{attribute 'OPC.UA.DA.StructuredType' := '1'}
FUNCTION_BLOCK FB_Unit_RO_RND EXTENDS FB_BaseDevice IMPLEMENTS I_Device

VAR
	bFirstRun: BOOL := TRUE;
	{attribute 'OPC.UA.DA' := '1'} 
	bOutContactor AT %Q*: BOOL := FALSE;
	
	
	{attribute 'OPC.UA.DA' := '0'} 
	eSMState: (WAIT, TURNING_ON, ON, TURNING_OFF, OFF);
	
	tDebounce: TIME := T#5S;
	fbTON_Debounce: TON := (PT := tDebounce, IN := FALSE);
	
END_VAR

fbTON_Debounce();

IF bFirstRun THEN
	fbTON_Debounce.IN := TRUE;
	bFirstRun := FALSE;
END_IF


IF GVL.bAutoUpdateDeviceState THEN
	eState := eStateTarget;	
END_IF


IF eMode = E_DeviceMode.MANUAL THEN
	bEnable := TRUE;
END_IF

IF bEnable AND eStateTarget = E_DeviceState.ON AND eState <> E_DeviceState.ON THEN
		eSMState := TURNING_ON;
END_IF

IF (bEnable = FALSE OR eStateTarget = E_DeviceState.OFF) AND eState <> E_DeviceState.OFF THEN
		eSMState := TURNING_OFF;
END_IF


CASE eSMState OF
	
	WAIT:
		//Wait for method call to change ESMState
		
	TURNING_ON: 
		IF fbTON_Debounce.Q THEN
			eState := E_DeviceState.TURNING_ON;
			bOutContactor := TRUE;
			fbTON_Debounce.IN := FALSE;
			eSMState := ON;
		END_IF

		
	ON:
		IF bOutContactor <> TRUE THEN
			raiseAlarm(Priority := E_AlarmPriority.High, Label := 'Power Lost', Enabled := TRUE, DeviceAlarmID := 1);
			eState := E_DeviceState.OFF;
			eSMState := TURNING_OFF;
		END_IF
			
	TURNING_OFF:
		fbTON_Debounce.IN := TRUE;
		bOutContactor := TRUE;
		eState := E_DeviceState.TURNING_OFF;
		bOutContactor := FALSE;
		eSMState := OFF;

	OFF:
		eState := E_DeviceState.OFF;
		eSMState := WAIT;
		fbTON_Debounce.IN := TRUE;
		
END_CASE

{warning 'add method implementation '}
METHOD disable : BOOL
bEnable := FALSE;
END_METHOD

{warning 'add method implementation '}
METHOD enable : BOOL
bEnable := TRUE;
END_METHOD

METHOD FB_init : BOOL
VAR_INPUT
	bInitRetains : BOOL; // if TRUE, the retain variables are initialized (warm start / cold start)
	bInCopyCode : BOOL;  // if TRUE, the instance afterwards gets moved into the copy code (online change)
	
	UnitID: STRING(80);
	UnitDescr: STRING(255); 
END_VAR
sID := UnitID;
sDescr := UnitDescr;
END_METHOD

METHOD setOff : BOOL
VAR_INPUT
END_VAR
eSMState := TURNING_OFF;
END_METHOD

METHOD setOn : BOOL
VAR_INPUT
END_VAR
eSMState := TURNING_ON;
END_METHOD

END_FUNCTION_BLOCK

(* stored: Version 1.1.0.1, ProductVersion 3.1.4024.12
   POU FB_Unit_RO_RND: Id {be8b5a2b-8843-42aa-8a40-21182057978c}, SpecialFunc None
   Method disable: Id {54656f00-5594-499d-bd42-c77bc73a0044}
   Method enable: Id {b2fa1289-5c77-45b7-9abb-82d67b098a30}
   Method FB_init: Id {e61bd435-9d8a-4e74-b194-9e33eac1d36d}
   Method setOff: Id {d3034f92-50a5-413b-983b-942e42fdebb6}
   Method setOn: Id {1729d636-cc5a-42b7-af0e-7e5a8c59d62f} *)
